(* CODESYS project ETML_DH10.library
   TcLibraryId: TE140x Module Vendor|ETML_DH10|0.0.0.9
   Company: TE140x Module Vendor
   Title: ETML_DH10
   Placeholder: ETML_DH10
   Version: 0.0.0.9

Project tree, tasks and I/O mapping:
  POUs/
    function block FB_ETML_DH10 [ST]: FB_exit, FB_init, nHResult, eInitExceptionHandling, eUpdateExceptionHandling, nExceptionCnt, stActiveException, bInitialized, bExecute
    TcCOM Wrapper/
      function block FB_ETML_DH10_TcCOM_InitStruct [ST]: FB_init, FB_afterinit, Reinit, FB_exit, eObjectState, nHResult, ipTcComObject, ipADI, nTaskOid, nTaskPriority, nTaskCycleTimeNs, nTaskPort, nTaskSortOrder, eTraceLevelMax, eModuleCaller, eCallerVerification, eStepSizeAdaptation, eExecutionSequence, bExecute, eAccessLockState, eInitExceptionHandling, eUpdateExceptionHandling, stModuleBuildInfo, bInitialized, nSkippedExecutionCount, stLibraryInfo, stModuleInfo, stModuleGeneratorInfo, stSimulinkModelInfo, eETML_DH10_P_Sharing, nETML_DH10_P_Definer, stETML_DH10_P, nCycleCount, nExceptionCount, stExceptionInfo
  DUTs/
    data type ST_FB_ETML_DH10_FB_Main
    data type ST_FB_ETML_DH10_FB_exit
    data type ST_FB_ETML_DH10_FB_init
    data type ST_GetSet_HRESULT
    data type E_FpExcptCtrlSetEx
    data type ST_GetSet_E_FpExcptCtrlSetEx
    data type ST_GetSet_ULINT
    data type ST_ExceptionInfo
    data type ST_GetSet_ST_ExceptionInfo
    data type ST_GetSet_BOOL
    data type ST_B_ETML_DH10_T
    data type ST_ExtU_ETML_DH10_T
    data type ST_ExtY_ETML_DH10_T
    data type ST_RT_MODEL_ETML_DH10_T
    data type ST_P_ETML_DH10_T
    data type E_ModuleCaller
    data type E_CallerVerification
    data type E_StepSizeAdaptation
    data type E_ExecutionSequence1
    data type E_FpExcptCtrlSet
    data type ST_TcMatSim_ModuleGeneratorInfo
    data type ST_TcMatSim_SimulinkModelInfo
    data type E_ParameterSharingType
    data type ST_FB_ETML_DH10_TcCOM_InitStruct
    data type ST_FB_ETML_DH10_TcCOM_InitStruct_FB_init
    data type ST_FB_ETML_DH10_TcCOM_InitStruct_FB_afterinit
    data type ST_FB_ETML_DH10_TcCOM_InitStruct_Reinit
    data type ST_FB_ETML_DH10_TcCOM_InitStruct_FB_Main
    data type ST_FB_ETML_DH10_TcCOM_InitStruct_FB_exit
    data type ST_GetSet_TCOM_STATE
    data type ST_GetSet_ITComObject
    data type ST_GetSet_ITcADI
    data type ST_ETML_DH10_U_T
    data type ST_ETML_DH10_Y_T
    data type ST_GetSet_OTCID
    data type ST_GetSet_UDINT
    data type ST_GetSet_UINT
    data type ST_GetSet_TcTraceLevel
    data type ST_GetSet_E_ModuleCaller
    data type ST_GetSet_E_CallerVerification
    data type ST_GetSet_E_StepSizeAdaptation
    data type ST_GetSet_E_ExecutionSequence1
    data type ST_GetSet_E_FpExcptCtrlSet
    data type ST_ModuleBuildInfo
    data type ST_GetSet_ST_ModuleBuildInfo
    data type ST_LibraryInfo
    data type ST_GetSet_ST_LibraryInfo
    data type ST_ModuleInfo
    data type ST_GetSet_ST_ModuleInfo
    data type ST_GetSet_ST_TcMatSim_ModuleGeneratorInfo
    data type ST_GetSet_ST_TcMatSim_SimulinkModelInfo
    data type ST_GetSet_E_ParameterSharingType
    data type ST_GetSet_ST_P_ETML_DH10_T
  Version/
    global variables Global_Version
*)

// DUTs/ST_FB_ETML_DH10_FB_Main
{attribute 'TcIecLibraryType'}
{attribute 'hide'}
TYPE ST_FB_ETML_DH10_FB_Main : 
	STRUCT
		{attribute 'GUID' := '18071995-0000-0000-0000-000000000018'}
		pInst : PVOID;
		result : BOOL;
		 {attribute 'hide'}
		_reserved1 : UINT_24_56;
	END_STRUCT
END_TYPE

// DUTs/ST_FB_ETML_DH10_FB_exit
{attribute 'TcIecLibraryType'}
{attribute 'hide'}
TYPE ST_FB_ETML_DH10_FB_exit : 
	STRUCT
		{attribute 'GUID' := '18071995-0000-0000-0000-000000000018'}
		pInst : PVOID;
		bInCopyCode : BOOL;
		result : BOOL;
		 {attribute 'hide'}
		_reserved1 : UINT_16_48;
	END_STRUCT
END_TYPE

// DUTs/ST_FB_ETML_DH10_FB_init
{attribute 'TcIecLibraryType'}
{attribute 'hide'}
TYPE ST_FB_ETML_DH10_FB_init : 
	STRUCT
		{attribute 'GUID' := '18071995-0000-0000-0000-000000000018'}
		pInst : PVOID;
		bInitRetains : BOOL;
		bInCopyCode : BOOL;
		result : BOOL;
		 {attribute 'hide'}
		_reserved1 : UINT_8_40;
	END_STRUCT
END_TYPE

// DUTs/ST_GetSet_HRESULT
{attribute 'TcIecLibraryType'}
{attribute 'hide'}
TYPE ST_GetSet_HRESULT : 
	STRUCT
		{attribute 'GUID' := '18071995-0000-0000-0000-000000000018'}
		pInst : PVOID;
		{attribute 'GUID' := '18071995-0000-0000-0000-000000000019'}
		nParam : HRESULT;
		 {attribute 'hide'}
		_reserved1 : UINT_0_32;
	END_STRUCT
END_TYPE

// DUTs/E_FpExcptCtrlSetEx
(* Generated from type 'TcMgSdk.FpExcptCtrlSetEx' *)
{attribute 'TcIecLibraryType'}
TYPE E_FpExcptCtrlSetEx : (
	CallerExceptions:=1, 	(* Use the floating point exception settings provided by the caller *)
	ThrowExceptions:=3, 	(* Enable floating point exceptions on invalid operations and divisions by zero *)
	SuppressExceptions:=13, 	(* Disable floating point exceptions. *)
	LogExceptions:=19, 	(* Log exception information. *)
	LogAndHold:=51, 	(* Log exception information and puase execution of the cyclic code after completion of the actual cycle *)
	LogAndCatch:=83, 	(* Log exception information and immediately terminate execution of the cyclic code. Reinitialization is required to restart. *)
	LogAndDump:=147, 	(* Log exception information, create a dump file with detailed exception information and try to continue execution of the cyclic code *)
	LogHoldAndDump:=179, 	(* Log exception information, create a dump file with detailed exception information and puase execution of the cyclic code after completion of the actual cycle *)
	LogCatchAndDump:=211	(* Log exception information, create a dump file with detailed exception information and immediately terminate execution of the cyclic code. Reinitialization is required to restart. *)
) USINT;
END_TYPE

// DUTs/ST_GetSet_E_FpExcptCtrlSetEx
{attribute 'TcIecLibraryType'}
{attribute 'hide'}
TYPE ST_GetSet_E_FpExcptCtrlSetEx : 
	STRUCT
		{attribute 'GUID' := '18071995-0000-0000-0000-000000000018'}
		pInst : PVOID;
		eParam : E_FpExcptCtrlSetEx;
		 {attribute 'hide'}
		_reserved1 : UINT_24_56;
	END_STRUCT
END_TYPE

// DUTs/ST_GetSet_ULINT
{attribute 'TcIecLibraryType'}
{attribute 'hide'}
TYPE ST_GetSet_ULINT : 
	STRUCT
		{attribute 'GUID' := '18071995-0000-0000-0000-000000000018'}
		pInst : PVOID;
		nParam : ULINT;
	END_STRUCT
END_TYPE

// DUTs/ST_ExceptionInfo
(* Generated from type 'TcMgSdk.ExceptionInfo' *)
{attribute 'TcIecLibraryType'}
TYPE ST_ExceptionInfo : 
	STRUCT
		(* Generated from item 'ExceptionCode' *)
		nExceptionCode : DINT;
		(* Generated from item 'TmxName' *)
		{attribute 'GUID' := '18071995-0000-0000-0000-00010000007F'}
		sTmxName : STRING(127);
		(* Generated from item 'TmxVersion' *)
		nTmxVersion : ARRAY [0..3] OF UDINT;
		(* Generated from item 'InstructionAddr' *)
		nInstructionAddr : UDINT;
		(* Generated from item 'ReturnAddr' *)
		nReturnAddr : ARRAY [0..3] OF UDINT;
		(* Generated from item 'DumpCreated' *)
		bDumpCreated : BOOL;
		 {attribute 'hide'}
		_reserved1 : ARRAY [1..3] OF USINT;
	END_STRUCT
END_TYPE

// DUTs/ST_GetSet_ST_ExceptionInfo
{attribute 'TcIecLibraryType'}
{attribute 'hide'}
TYPE ST_GetSet_ST_ExceptionInfo : 
	STRUCT
		{attribute 'GUID' := '18071995-0000-0000-0000-000000000018'}
		pInst : PVOID;
		stParam : ST_ExceptionInfo;
		 {attribute 'hide'}
		_reserved1 : UINT_0_32;
	END_STRUCT
END_TYPE

// DUTs/ST_GetSet_BOOL
{attribute 'TcIecLibraryType'}
{attribute 'hide'}
TYPE ST_GetSet_BOOL : 
	STRUCT
		{attribute 'GUID' := '18071995-0000-0000-0000-000000000018'}
		pInst : PVOID;
		bParam : BOOL;
		 {attribute 'hide'}
		_reserved1 : UINT_24_56;
	END_STRUCT
END_TYPE

// DUTs/ST_B_ETML_DH10_T
(* Generated from type 'B_ETML_DH10_T' *)
{attribute 'TcIecLibraryType'}
TYPE ST_B_ETML_DH10_T : 
	STRUCT
		(* Generated from item 'Sum4' *)
		fSum4 : LREAL;
		(* Generated from item 'Sum5' *)
		fSum5 : LREAL;
		(* Generated from item 'Sum4_g' *)
		fSum4_g : LREAL;
		(* Generated from item 'Sum5_o' *)
		fSum5_o : LREAL;
		(* Generated from item 'Sum4_k' *)
		fSum4_k : LREAL;
		(* Generated from item 'Sum5_c' *)
		fSum5_c : LREAL;
		(* Generated from item 'Sum4_n' *)
		fSum4_n : LREAL;
		(* Generated from item 'Sum5_m' *)
		fSum5_m : LREAL;
		(* Generated from item 'Sum4_c' *)
		fSum4_c : LREAL;
		(* Generated from item 'Sum5_l' *)
		fSum5_l : LREAL;
		(* Generated from item 'Sum4_j' *)
		fSum4_j : LREAL;
		(* Generated from item 'Sum5_p' *)
		fSum5_p : LREAL;
		(* Generated from item 'Sum4_nw' *)
		fSum4_nw : LREAL;
		(* Generated from item 'Sum5_d' *)
		fSum5_d : LREAL;
		(* Generated from item 'Sum4_gt' *)
		fSum4_gt : LREAL;
		(* Generated from item 'Sum5_ob' *)
		fSum5_ob : LREAL;
		(* Generated from item 'q' *)
		fq : LREAL;
		(* Generated from item 'q_g' *)
		fq_g : LREAL;
		(* Generated from item 'q_gi' *)
		fq_gi : LREAL;
		(* Generated from item 'UnaryMinus' *)
		fUnaryMinus : LREAL;
		(* Generated from item 'UnaryMinus_n' *)
		fUnaryMinus_n : LREAL;
		(* Generated from item 'UnaryMinus_o' *)
		fUnaryMinus_o : LREAL;
		(* Generated from item 'UnaryMinus_k' *)
		fUnaryMinus_k : LREAL;
		(* Generated from item 'UnaryMinus_f' *)
		fUnaryMinus_f : LREAL;
		(* Generated from item 'UnaryMinus_l' *)
		fUnaryMinus_l : LREAL;
		(* Generated from item 'UnaryMinus_g' *)
		fUnaryMinus_g : LREAL;
		(* Generated from item 'UnaryMinus_d' *)
		fUnaryMinus_d : LREAL;
		(* Generated from item 's' *)
		fs : LREAL;
		(* Generated from item 's_m' *)
		fs_m : LREAL;
		(* Generated from item 's_h' *)
		fs_h : LREAL;
		(* Generated from item 's_e' *)
		fs_e : LREAL;
		(* Generated from item 's_c' *)
		fs_c : LREAL;
		(* Generated from item 's_l' *)
		fs_l : LREAL;
		(* Generated from item 's_d' *)
		fs_d : LREAL;
		(* Generated from item 's_du' *)
		fs_du : LREAL;
		(* Generated from item 'u' *)
		fu : LREAL;
		(* Generated from item 'Add5' *)
		fAdd5 : LREAL;
		(* Generated from item 'Product4' *)
		fProduct4 : LREAL;
		(* Generated from item 'u_c' *)
		fu_c : LREAL;
		(* Generated from item 'Add5_m' *)
		fAdd5_m : LREAL;
		(* Generated from item 'Product4_p' *)
		fProduct4_p : LREAL;
		(* Generated from item 'u_a' *)
		fu_a : LREAL;
		(* Generated from item 'Add5_j' *)
		fAdd5_j : LREAL;
		(* Generated from item 'Product4_g' *)
		fProduct4_g : LREAL;
		(* Generated from item 'u_l' *)
		fu_l : LREAL;
		(* Generated from item 'Add5_b' *)
		fAdd5_b : LREAL;
		(* Generated from item 'u_m' *)
		fu_m : LREAL;
		(* Generated from item 'Product4_c' *)
		fProduct4_c : LREAL;
		(* Generated from item 'u_o' *)
		fu_o : LREAL;
		(* Generated from item 'Product4_k' *)
		fProduct4_k : LREAL;
		(* Generated from item 'u_g' *)
		fu_g : LREAL;
		(* Generated from item 'Product4_d' *)
		fProduct4_d : LREAL;
		(* Generated from item 'u_p' *)
		fu_p : LREAL;
		(* Generated from item 'Add5_bw' *)
		fAdd5_bw : LREAL;
		(* Generated from item 'Product4_h' *)
		fProduct4_h : LREAL;
		(* Generated from item 'Product1' *)
		fProduct1 : LREAL;
		(* Generated from item 'Product1_e' *)
		fProduct1_e : LREAL;
		(* Generated from item 'Sum2' *)
		fSum2 : LREAL;
		(* Generated from item 'Product1_m' *)
		fProduct1_m : LREAL;
		(* Generated from item 'Sum2_i' *)
		fSum2_i : LREAL;
		(* Generated from item 'Product1_m4' *)
		fProduct1_m4 : LREAL;
		(* Generated from item 'Sum2_j' *)
		fSum2_j : LREAL;
		(* Generated from item 'Product1_f' *)
		fProduct1_f : LREAL;
		(* Generated from item 'UnitDelay2' *)
		fUnitDelay2 : LREAL;
		(* Generated from item 'Product1_l' *)
		fProduct1_l : LREAL;
		(* Generated from item 'UnitDelay2_p' *)
		fUnitDelay2_p : LREAL;
		(* Generated from item 'Product1_a' *)
		fProduct1_a : LREAL;
		(* Generated from item 'UnitDelay2_i' *)
		fUnitDelay2_i : LREAL;
		(* Generated from item 'Product1_o' *)
		fProduct1_o : LREAL;
		(* Generated from item 'Product3' *)
		fProduct3 : LREAL;
		(* Generated from item 'UnitDelay2_l' *)
		fUnitDelay2_l : LREAL;
		(* Generated from item 'Product3_e' *)
		fProduct3_e : LREAL;
		(* Generated from item 'Product3_j' *)
		fProduct3_j : LREAL;
		(* Generated from item 'Product3_a' *)
		fProduct3_a : LREAL;
		(* Generated from item 'Product3_c' *)
		fProduct3_c : LREAL;
		(* Generated from item 'UnitDelay2_k' *)
		fUnitDelay2_k : LREAL;
		(* Generated from item 'Product4_f' *)
		fProduct4_f : LREAL;
		(* Generated from item 'Product3_i' *)
		fProduct3_i : LREAL;
		(* Generated from item 'Product3_o' *)
		fProduct3_o : LREAL;
		(* Generated from item 'Product3_ao' *)
		fProduct3_ao : LREAL;
		(* Generated from item 'RelationalOperator' *)
		bRelationalOperator : BOOL;
		 {attribute 'hide'}
		_reserved1 : ARRAY [1..7] OF USINT;
	END_STRUCT
END_TYPE

// DUTs/ST_ExtU_ETML_DH10_T
(* Generated from type 'ExtU_ETML_DH10_T' *)
{attribute 'TcIecLibraryType'}
TYPE ST_ExtU_ETML_DH10_T : 
	STRUCT
		(* Generated from item 'OffsetLeft' *)
		fOffsetLeft : LREAL;
		(* Generated from item 'OffsetRight' *)
		fOffsetRight : LREAL;
	END_STRUCT
END_TYPE

// DUTs/ST_ExtY_ETML_DH10_T
(* Generated from type 'ExtY_ETML_DH10_T' *)
{attribute 'TcIecLibraryType'}
TYPE ST_ExtY_ETML_DH10_T : 
	STRUCT
		(* Generated from item 'CurrentAngleLeft' *)
		fCurrentAngleLeft : LREAL;
		(* Generated from item 'CurrentAngleRight' *)
		fCurrentAngleRight : LREAL;
	END_STRUCT
END_TYPE

// DUTs/ST_RT_MODEL_ETML_DH10_T
(* Generated from type 'RT_MODEL_ETML_DH10_T' *)
{attribute 'TcIecLibraryType'}
TYPE ST_RT_MODEL_ETML_DH10_T : 
	STRUCT
		errorStatus : POINTER TO SINT;
		blockIO : POINTER TO ST_B_ETML_DH10_T;
		inputs : POINTER TO ST_ExtU_ETML_DH10_T;
		outputs : POINTER TO ST_ExtY_ETML_DH10_T;
	END_STRUCT
END_TYPE

// DUTs/ST_P_ETML_DH10_T
(* Generated from type 'P_ETML_DH10_T' *)
{attribute 'TcIecLibraryType'}
TYPE ST_P_ETML_DH10_T : 
	STRUCT
		(* Generated from item 'ETML_gain_left' *)
		fETML_gain_left : LREAL;
		(* Generated from item 'ETML_gain_right' *)
		fETML_gain_right : LREAL;
		(* Generated from item 'ETML_power_constant' *)
		fETML_power_constant : LREAL;
		(* Generated from item 'f_ETML_notch_main_1' *)
		ff_ETML_notch_main_1 : LREAL;
		(* Generated from item 'f_ETML_notch_main_2' *)
		ff_ETML_notch_main_2 : LREAL;
		(* Generated from item 'f_ETML_notch_main_3' *)
		ff_ETML_notch_main_3 : LREAL;
		(* Generated from item 'f_ETML_notch_main_4' *)
		ff_ETML_notch_main_4 : LREAL;
		(* Generated from item 'notch_damp' *)
		fnotch_damp : LREAL;
		(* Generated from item 'notch_gmin' *)
		fnotch_gmin : LREAL;
		(* Generated from item 'enable_ETML_main_notch_1' *)
		benable_ETML_main_notch_1 : BOOL;
		(* Generated from item 'enable_ETML_main_notch_2' *)
		benable_ETML_main_notch_2 : BOOL;
		(* Generated from item 'enable_ETML_main_notch_3' *)
		benable_ETML_main_notch_3 : BOOL;
		(* Generated from item 'enable_ETML_main_notch_4' *)
		benable_ETML_main_notch_4 : BOOL;
		 {attribute 'hide'}
		_reserved1 : UDINT;
		(* Generated from item 'Constant2_Value' *)
		fConstant2_Value : LREAL;
		(* Generated from item 'Constant_Value' *)
		fConstant_Value : LREAL;
		(* Generated from item 'tau_Gain' *)
		ftau_Gain : LREAL;
		(* Generated from item 'Bias_Bias' *)
		fBias_Bias : LREAL;
		(* Generated from item 'two_Gain' *)
		ftwo_Gain : LREAL;
		(* Generated from item 'one_Gain' *)
		fone_Gain : LREAL;
		(* Generated from item 'UnitDelay1_InitialCondition' *)
		fUnitDelay1_InitialCondition : LREAL;
		(* Generated from item 'tau_Gain_n' *)
		ftau_Gain_n : LREAL;
		(* Generated from item 'Bias_Bias_e' *)
		fBias_Bias_e : LREAL;
		(* Generated from item 'two_Gain_i' *)
		ftwo_Gain_i : LREAL;
		(* Generated from item 'one_Gain_k' *)
		fone_Gain_k : LREAL;
		(* Generated from item 'UnitDelay1_InitialCondition_p' *)
		fUnitDelay1_InitialCondition_p : LREAL;
		(* Generated from item 'tau_Gain_j' *)
		ftau_Gain_j : LREAL;
		(* Generated from item 'Bias_Bias_h' *)
		fBias_Bias_h : LREAL;
		(* Generated from item 'two_Gain_b' *)
		ftwo_Gain_b : LREAL;
		(* Generated from item 'one_Gain_e' *)
		fone_Gain_e : LREAL;
		(* Generated from item 'UnitDelay1_InitialCondition_b' *)
		fUnitDelay1_InitialCondition_b : LREAL;
		(* Generated from item 'tau_Gain_k' *)
		ftau_Gain_k : LREAL;
		(* Generated from item 'Bias_Bias_a' *)
		fBias_Bias_a : LREAL;
		(* Generated from item 'two_Gain_h' *)
		ftwo_Gain_h : LREAL;
		(* Generated from item 'one_Gain_ea' *)
		fone_Gain_ea : LREAL;
		(* Generated from item 'UnitDelay1_InitialCondition_d' *)
		fUnitDelay1_InitialCondition_d : LREAL;
		(* Generated from item 'Left_UpperSat' *)
		fLeft_UpperSat : LREAL;
		(* Generated from item 'Left_LowerSat' *)
		fLeft_LowerSat : LREAL;
		(* Generated from item 'tau_Gain_l' *)
		ftau_Gain_l : LREAL;
		(* Generated from item 'Bias_Bias_j' *)
		fBias_Bias_j : LREAL;
		(* Generated from item 'two_Gain_o' *)
		ftwo_Gain_o : LREAL;
		(* Generated from item 'one_Gain_o' *)
		fone_Gain_o : LREAL;
		(* Generated from item 'UnitDelay1_InitialCondition_j' *)
		fUnitDelay1_InitialCondition_j : LREAL;
		(* Generated from item 'tau_Gain_f' *)
		ftau_Gain_f : LREAL;
		(* Generated from item 'Bias_Bias_b' *)
		fBias_Bias_b : LREAL;
		(* Generated from item 'two_Gain_c' *)
		ftwo_Gain_c : LREAL;
		(* Generated from item 'one_Gain_l' *)
		fone_Gain_l : LREAL;
		(* Generated from item 'UnitDelay1_InitialCondition_a' *)
		fUnitDelay1_InitialCondition_a : LREAL;
		(* Generated from item 'tau_Gain_lc' *)
		ftau_Gain_lc : LREAL;
		(* Generated from item 'Bias_Bias_i' *)
		fBias_Bias_i : LREAL;
		(* Generated from item 'two_Gain_m' *)
		ftwo_Gain_m : LREAL;
		(* Generated from item 'one_Gain_ef' *)
		fone_Gain_ef : LREAL;
		(* Generated from item 'UnitDelay1_InitialCondition_d5' *)
		fUnitDelay1_InitialCondition_d5 : LREAL;
		(* Generated from item 'tau_Gain_e' *)
		ftau_Gain_e : LREAL;
		(* Generated from item 'Bias_Bias_l' *)
		fBias_Bias_l : LREAL;
		(* Generated from item 'two_Gain_it' *)
		ftwo_Gain_it : LREAL;
		(* Generated from item 'one_Gain_a' *)
		fone_Gain_a : LREAL;
		(* Generated from item 'UnitDelay1_InitialCondition_l' *)
		fUnitDelay1_InitialCondition_l : LREAL;
		(* Generated from item 'Right_UpperSat' *)
		fRight_UpperSat : LREAL;
		(* Generated from item 'Right_LowerSat' *)
		fRight_LowerSat : LREAL;
		(* Generated from item 'Bias1_Bias' *)
		fBias1_Bias : LREAL;
		(* Generated from item 'Gain_Gain' *)
		fGain_Gain : LREAL;
		(* Generated from item 'UnitDelay2_InitialCondition' *)
		fUnitDelay2_InitialCondition : LREAL;
		(* Generated from item 'Bias1_Bias_b' *)
		fBias1_Bias_b : LREAL;
		(* Generated from item 'Gain_Gain_g' *)
		fGain_Gain_g : LREAL;
		(* Generated from item 'UnitDelay2_InitialCondition_p' *)
		fUnitDelay2_InitialCondition_p : LREAL;
		(* Generated from item 'Bias1_Bias_n' *)
		fBias1_Bias_n : LREAL;
		(* Generated from item 'Gain_Gain_k' *)
		fGain_Gain_k : LREAL;
		(* Generated from item 'UnitDelay2_InitialCondition_o' *)
		fUnitDelay2_InitialCondition_o : LREAL;
		(* Generated from item 'Bias1_Bias_c' *)
		fBias1_Bias_c : LREAL;
		(* Generated from item 'Gain_Gain_e' *)
		fGain_Gain_e : LREAL;
		(* Generated from item 'UnitDelay2_InitialCondition_f' *)
		fUnitDelay2_InitialCondition_f : LREAL;
		(* Generated from item 'Bias1_Bias_l' *)
		fBias1_Bias_l : LREAL;
		(* Generated from item 'Gain_Gain_ey' *)
		fGain_Gain_ey : LREAL;
		(* Generated from item 'UnitDelay2_InitialCondition_k' *)
		fUnitDelay2_InitialCondition_k : LREAL;
		(* Generated from item 'Bias1_Bias_j' *)
		fBias1_Bias_j : LREAL;
		(* Generated from item 'Gain_Gain_ky' *)
		fGain_Gain_ky : LREAL;
		(* Generated from item 'UnitDelay2_InitialCondition_l' *)
		fUnitDelay2_InitialCondition_l : LREAL;
		(* Generated from item 'Bias1_Bias_d' *)
		fBias1_Bias_d : LREAL;
		(* Generated from item 'Gain_Gain_f' *)
		fGain_Gain_f : LREAL;
		(* Generated from item 'UnitDelay2_InitialCondition_n' *)
		fUnitDelay2_InitialCondition_n : LREAL;
		(* Generated from item 'Bias1_Bias_cn' *)
		fBias1_Bias_cn : LREAL;
		(* Generated from item 'Gain_Gain_h' *)
		fGain_Gain_h : LREAL;
		(* Generated from item 'UnitDelay2_InitialCondition_i' *)
		fUnitDelay2_InitialCondition_i : LREAL;
	END_STRUCT
END_TYPE

// DUTs/E_ModuleCaller
(* Generated from type 'TcMgSdk.ModuleCaller' *)
{attribute 'TcIecLibraryType'}
TYPE E_ModuleCaller : (
	CyclicTask:=0, 	(* Add to the specified cyclic caller tasks. *)
	Module:=1	(* Don't add to cyclic callers. The module can be called from other TwinCAT modules (e. g. a PLC). *)
) DINT;
END_TYPE

// DUTs/E_CallerVerification
(* Generated from type 'TcMgSdk.CallerVerification' *)
{attribute 'TcIecLibraryType'}
TYPE E_CallerVerification : (
	Default:=0, 	(* Verify the caller task only if the "ModuleCaller" parameter is set to "Module" but not when added to cyclic caller tasks. *)
	Always:=1, 	(* Always verify the caller context to prevent concurrent execution of model code and corresponding DataArea mappings. *)
	Never:=2	(* Skip caller verification to reduce execution times. *)
) DINT;
END_TYPE

// DUTs/E_StepSizeAdaptation
(* Generated from type 'TcMgSdk.StepSizeAdaptation' *)
{attribute 'TcIecLibraryType'}
TYPE E_StepSizeAdaptation : (
	RequireMatchingTaskCycleTime:=0, 	(* Don't accept task cycle times other than the Simulink step sizes. *)
	UseTaskCycleTime:=1, 	(* Adapt the Smulink step sizes to the task cycle times. *)
	UseModelStepSize:=2	(* Keep the Smulink step sizes, independent of the callers cycle time. *)
) DINT;
END_TYPE

// DUTs/E_ExecutionSequence1
(* Generated from type 'TcMgSdk.ExecutionSequence1' *)
{attribute 'TcIecLibraryType'}
TYPE E_ExecutionSequence1 : (
	UpdateBeforeOutputMapping:=0, 	(* Input mapping -> State and output update -> Output mapping -> ADS processing *)
	IoAtTaskBegin:=1	(* Input mapping -> Code execution -> Output update -> ADS processing *)
) DINT;
END_TYPE

// DUTs/E_FpExcptCtrlSet
(* Generated from type 'TcMgSdk.FpExcptCtrlSet' *)
{attribute 'TcIecLibraryType'}
TYPE E_FpExcptCtrlSet : (
	CallerExceptions:=1, 	(* Use the floating point exception settings provided by the caller *)
	ThrowExceptions:=3, 	(* Enable floating point exceptions on invalid operations and divisions by zero *)
	SuppressExceptions:=5	(* Disable floating point exceptions. *)
) USINT;
END_TYPE

// DUTs/ST_TcMatSim_ModuleGeneratorInfo
(* Generated from type 'TcMatSim.ModuleGeneratorInfo' *)
{attribute 'TcIecLibraryType'}
TYPE ST_TcMatSim_ModuleGeneratorInfo : 
	STRUCT
		(* Generated from item 'MatlabVersion' *)
		nMatlabVersion : ARRAY [0..3] OF UDINT;
		(* Generated from item 'TE140xVersion' *)
		nTE140xVersion : ARRAY [0..3] OF UDINT;
	END_STRUCT
END_TYPE

// DUTs/ST_TcMatSim_SimulinkModelInfo
(* Generated from type 'TcMatSim.SimulinkModelInfo' *)
{attribute 'TcIecLibraryType'}
TYPE ST_TcMatSim_SimulinkModelInfo : 
	STRUCT
		(* Generated from item 'ModelName' *)
		{attribute 'GUID' := '18071995-0000-0000-0000-00010000007F'}
		sModelName : STRING(127);
		(* Generated from item 'SimulinkVersion' *)
		nSimulinkVersion : ARRAY [0..3] OF UDINT;
		(* Generated from item 'ModelVersion' *)
		nModelVersion : ARRAY [0..3] OF UDINT;
		(* Generated from item 'ModelChecksum' *)
		nModelChecksum : ARRAY [0..3] OF UDINT;
	END_STRUCT
END_TYPE

// DUTs/E_ParameterSharingType
(* Generated from type 'ParameterSharingType' *)
{attribute 'TcIecLibraryType'}
TYPE E_ParameterSharingType : (
	Define:=0, 	(* This module instance defines the parameter values for all further instances of this module class. Exactly one instance of this module class must use this option. *)
	Inherit:=1	(* This module instance inherits the parameter values from the instance of this module class configured to "Define" the parameter values. Model parameters configured at this instsance are ignored. *)
) DINT;
END_TYPE

// DUTs/ST_FB_ETML_DH10_TcCOM_InitStruct
{attribute 'TcIecLibraryType'}
TYPE ST_FB_ETML_DH10_TcCOM_InitStruct : 
	STRUCT
		{attribute 'GUID' := '18071995-0000-0000-0000-000000000061'}
		eObjState : TCOM_STATE := TCOM_STATE.TCOM_STATE_OP;
		{attribute 'GUID' := '18071995-0000-0000-0000-00010000007F'}
		sObjName : STRING(127);
		{attribute 'GUID' := '18071995-0000-0000-0000-00000000000F'}
		nOid : OTCID := 4294967295;
		{attribute 'GUID' := '18071995-0000-0000-0000-00000000000F'}
		nTaskOid : OTCID;
		nTaskSortOrder : UDINT;
		{attribute 'GUID' := '8007AE3B-86BB-40F2-B385-EF87FCC239A4'}
		eTraceLevelMax : TcTraceLevel := TcTraceLevel.tlInfo;
		eModuleCaller : E_ModuleCaller := E_ModuleCaller.CyclicTask;
		eCallerVerification : E_CallerVerification := E_CallerVerification.Default;
		eStepSizeAdaptation : E_StepSizeAdaptation := E_StepSizeAdaptation.RequireMatchingTaskCycleTime;
		eExecutionSequence : E_ExecutionSequence1 := E_ExecutionSequence1.UpdateBeforeOutputMapping;
		bExecute : BOOL := TRUE;
		 {attribute 'hide'}
		_reserved1 : ARRAY [1..3] OF USINT;
		{attribute 'GUID' := '18071995-0000-0000-0000-000000000061'}
		eAccessLockState : TCOM_STATE := TCOM_STATE.TCOM_STATE_OP;
		eInitExceptionHandling : E_FpExcptCtrlSet := E_FpExcptCtrlSet.CallerExceptions;
		eUpdateExceptionHandling : E_FpExcptCtrlSetEx := E_FpExcptCtrlSetEx.CallerExceptions;
		 {attribute 'hide'}
		_reserved2 : UINT;
		stModuleGeneratorInfo : ST_TcMatSim_ModuleGeneratorInfo;
		stSimulinkModelInfo : ST_TcMatSim_SimulinkModelInfo;
		eETML_DH10_P_Sharing : E_ParameterSharingType := E_ParameterSharingType.Define;
		 {attribute 'hide'}
		_reserved3 : UDINT;
		stETML_DH10_P : ST_P_ETML_DH10_T := (fETML_gain_left := 16.91503741, fETML_gain_right := 16.91503741, fETML_power_constant := 0.46047809, ff_ETML_notch_main_1 := 0, ff_ETML_notch_main_2 := 0, ff_ETML_notch_main_3 := 0, ff_ETML_notch_main_4 := 0, fnotch_damp := 0.3, fnotch_gmin := 0.1, benable_ETML_main_notch_1 := FALSE, benable_ETML_main_notch_2 := FALSE, benable_ETML_main_notch_3 := FALSE, benable_ETML_main_notch_4 := FALSE, fConstant2_Value := 45, fConstant_Value := 0, ftau_Gain := 0.003, fBias_Bias := 1, ftwo_Gain := 2, fone_Gain := 1, fUnitDelay1_InitialCondition := 0, ftau_Gain_n := 0.003, fBias_Bias_e := 1, ftwo_Gain_i := 2, fone_Gain_k := 1, fUnitDelay1_InitialCondition_p := 0, ftau_Gain_j := 0.003, fBias_Bias_h := 1, ftwo_Gain_b := 2, fone_Gain_e := 1, fUnitDelay1_InitialCondition_b := 0, ftau_Gain_k := 0.003, fBias_Bias_a := 1, ftwo_Gain_h := 2, fone_Gain_ea := 1, fUnitDelay1_InitialCondition_d := 0, fLeft_UpperSat := 90, fLeft_LowerSat := 0, ftau_Gain_l := 0.003, fBias_Bias_j := 1, ftwo_Gain_o := 2, fone_Gain_o := 1, fUnitDelay1_InitialCondition_j := 0, ftau_Gain_f := 0.003, fBias_Bias_b := 1, ftwo_Gain_c := 2, fone_Gain_l := 1, fUnitDelay1_InitialCondition_a := 0, ftau_Gain_lc := 0.003, fBias_Bias_i := 1, ftwo_Gain_m := 2, fone_Gain_ef := 1, fUnitDelay1_InitialCondition_d5 := 0, ftau_Gain_e := 0.003, fBias_Bias_l := 1, ftwo_Gain_it := 2, fone_Gain_a := 1, fUnitDelay1_InitialCondition_l := 0, fRight_UpperSat := 90, fRight_LowerSat := 0, fBias1_Bias := 1, fGain_Gain := 2, fUnitDelay2_InitialCondition := 0, fBias1_Bias_b := 1, fGain_Gain_g := 2, fUnitDelay2_InitialCondition_p := 0, fBias1_Bias_n := 1, fGain_Gain_k := 2, fUnitDelay2_InitialCondition_o := 0, fBias1_Bias_c := 1, fGain_Gain_e := 2, fUnitDelay2_InitialCondition_f := 0, fBias1_Bias_l := 1, fGain_Gain_ey := 2, fUnitDelay2_InitialCondition_k := 0, fBias1_Bias_j := 1, fGain_Gain_ky := 2, fUnitDelay2_InitialCondition_l := 0, fBias1_Bias_d := 1, fGain_Gain_f := 2, fUnitDelay2_InitialCondition_n := 0, fBias1_Bias_cn := 1, fGain_Gain_h := 2, fUnitDelay2_InitialCondition_i := 0);
	END_STRUCT
END_TYPE

// DUTs/ST_FB_ETML_DH10_TcCOM_InitStruct_FB_init
{attribute 'TcIecLibraryType'}
{attribute 'hide'}
TYPE ST_FB_ETML_DH10_TcCOM_InitStruct_FB_init : 
	STRUCT
		{attribute 'GUID' := '18071995-0000-0000-0000-000000000018'}
		pInst : PVOID;
		bInitRetains : BOOL;
		bInCopyCode : BOOL;
		 {attribute 'hide'}
		_reserved1 : UINT_16_48;
		stInit : REFERENCE TO ST_FB_ETML_DH10_TcCOM_InitStruct;
		result : BOOL;
		 {attribute 'hide'}
		_reserved2 : UINT_24_56;
	END_STRUCT
END_TYPE

// DUTs/ST_FB_ETML_DH10_TcCOM_InitStruct_FB_afterinit
{attribute 'TcIecLibraryType'}
{attribute 'hide'}
TYPE ST_FB_ETML_DH10_TcCOM_InitStruct_FB_afterinit : 
	STRUCT
		{attribute 'GUID' := '18071995-0000-0000-0000-000000000018'}
		pInst : PVOID;
		result : BOOL;
		 {attribute 'hide'}
		_reserved1 : UINT_24_56;
	END_STRUCT
END_TYPE

// DUTs/ST_FB_ETML_DH10_TcCOM_InitStruct_Reinit
{attribute 'TcIecLibraryType'}
{attribute 'hide'}
TYPE ST_FB_ETML_DH10_TcCOM_InitStruct_Reinit : 
	STRUCT
		{attribute 'GUID' := '18071995-0000-0000-0000-000000000018'}
		pInst : PVOID;
		stReInit : ST_FB_ETML_DH10_TcCOM_InitStruct;
		result : BOOL;
		 {attribute 'hide'}
		_reserved1 : ARRAY [1..7] OF USINT;
	END_STRUCT
END_TYPE

// DUTs/ST_FB_ETML_DH10_TcCOM_InitStruct_FB_Main
{attribute 'TcIecLibraryType'}
{attribute 'hide'}
TYPE ST_FB_ETML_DH10_TcCOM_InitStruct_FB_Main : 
	STRUCT
		{attribute 'GUID' := '18071995-0000-0000-0000-000000000018'}
		pInst : PVOID;
		result : BOOL;
		 {attribute 'hide'}
		_reserved1 : UINT_24_56;
	END_STRUCT
END_TYPE

// DUTs/ST_FB_ETML_DH10_TcCOM_InitStruct_FB_exit
{attribute 'TcIecLibraryType'}
{attribute 'hide'}
TYPE ST_FB_ETML_DH10_TcCOM_InitStruct_FB_exit : 
	STRUCT
		{attribute 'GUID' := '18071995-0000-0000-0000-000000000018'}
		pInst : PVOID;
		bInCopyCode : BOOL;
		result : BOOL;
		 {attribute 'hide'}
		_reserved1 : UINT_16_48;
	END_STRUCT
END_TYPE

// DUTs/ST_GetSet_TCOM_STATE
{attribute 'TcIecLibraryType'}
{attribute 'hide'}
TYPE ST_GetSet_TCOM_STATE : 
	STRUCT
		{attribute 'GUID' := '18071995-0000-0000-0000-000000000018'}
		pInst : PVOID;
		{attribute 'GUID' := '18071995-0000-0000-0000-000000000061'}
		eParam : TCOM_STATE;
		 {attribute 'hide'}
		_reserved1 : UINT_0_32;
	END_STRUCT
END_TYPE

// DUTs/ST_GetSet_ITComObject
{attribute 'TcIecLibraryType'}
{attribute 'hide'}
TYPE ST_GetSet_ITComObject : 
	STRUCT
		{attribute 'GUID' := '18071995-0000-0000-0000-000000000018'}
		pInst : PVOID;
		{attribute 'GUID' := '00000012-0000-0000-E000-000000000064'}
		ipParam : ITComObject;
	END_STRUCT
END_TYPE

// DUTs/ST_GetSet_ITcADI
{attribute 'TcIecLibraryType'}
{attribute 'hide'}
TYPE ST_GetSet_ITcADI : 
	STRUCT
		{attribute 'GUID' := '18071995-0000-0000-0000-000000000018'}
		pInst : PVOID;
		{attribute 'GUID' := '03000012-0000-0000-E000-000000000064'}
		ipParam : ITcADI;
	END_STRUCT
END_TYPE

// DUTs/ST_ETML_DH10_U_T
(* Generated from type 'ETML_DH10_U_T' *)
{attribute 'TcIecLibraryType'}
TYPE ST_ETML_DH10_U_T : 
	STRUCT
		(* Generated from item 'OffsetLeft' *)
		fOffsetLeft : LREAL;
		(* Generated from item 'OffsetRight' *)
		fOffsetRight : LREAL;
	END_STRUCT
END_TYPE

// DUTs/ST_ETML_DH10_Y_T
(* Generated from type 'ETML_DH10_Y_T' *)
{attribute 'TcIecLibraryType'}
TYPE ST_ETML_DH10_Y_T : 
	STRUCT
		(* Generated from item 'CurrentAngleLeft' *)
		fCurrentAngleLeft : LREAL;
		(* Generated from item 'CurrentAngleRight' *)
		fCurrentAngleRight : LREAL;
	END_STRUCT
END_TYPE

// DUTs/ST_GetSet_OTCID
{attribute 'TcIecLibraryType'}
{attribute 'hide'}
TYPE ST_GetSet_OTCID : 
	STRUCT
		{attribute 'GUID' := '18071995-0000-0000-0000-000000000018'}
		pInst : PVOID;
		{attribute 'GUID' := '18071995-0000-0000-0000-00000000000F'}
		nParam : OTCID;
		 {attribute 'hide'}
		_reserved1 : UINT_0_32;
	END_STRUCT
END_TYPE

// DUTs/ST_GetSet_UDINT
{attribute 'TcIecLibraryType'}
{attribute 'hide'}
TYPE ST_GetSet_UDINT : 
	STRUCT
		{attribute 'GUID' := '18071995-0000-0000-0000-000000000018'}
		pInst : PVOID;
		nParam : UDINT;
		 {attribute 'hide'}
		_reserved1 : UINT_0_32;
	END_STRUCT
END_TYPE

// DUTs/ST_GetSet_UINT
{attribute 'TcIecLibraryType'}
{attribute 'hide'}
TYPE ST_GetSet_UINT : 
	STRUCT
		{attribute 'GUID' := '18071995-0000-0000-0000-000000000018'}
		pInst : PVOID;
		nParam : UINT;
		 {attribute 'hide'}
		_reserved1 : UINT_16_48;
	END_STRUCT
END_TYPE

// DUTs/ST_GetSet_TcTraceLevel
{attribute 'TcIecLibraryType'}
{attribute 'hide'}
TYPE ST_GetSet_TcTraceLevel : 
	STRUCT
		{attribute 'GUID' := '18071995-0000-0000-0000-000000000018'}
		pInst : PVOID;
		{attribute 'GUID' := '8007AE3B-86BB-40F2-B385-EF87FCC239A4'}
		eParam : TcTraceLevel;
		 {attribute 'hide'}
		_reserved1 : UINT_0_32;
	END_STRUCT
END_TYPE

// DUTs/ST_GetSet_E_ModuleCaller
{attribute 'TcIecLibraryType'}
{attribute 'hide'}
TYPE ST_GetSet_E_ModuleCaller : 
	STRUCT
		{attribute 'GUID' := '18071995-0000-0000-0000-000000000018'}
		pInst : PVOID;
		eParam : E_ModuleCaller;
		 {attribute 'hide'}
		_reserved1 : UINT_0_32;
	END_STRUCT
END_TYPE

// DUTs/ST_GetSet_E_CallerVerification
{attribute 'TcIecLibraryType'}
{attribute 'hide'}
TYPE ST_GetSet_E_CallerVerification : 
	STRUCT
		{attribute 'GUID' := '18071995-0000-0000-0000-000000000018'}
		pInst : PVOID;
		eParam : E_CallerVerification;
		 {attribute 'hide'}
		_reserved1 : UINT_0_32;
	END_STRUCT
END_TYPE

// DUTs/ST_GetSet_E_StepSizeAdaptation
{attribute 'TcIecLibraryType'}
{attribute 'hide'}
TYPE ST_GetSet_E_StepSizeAdaptation : 
	STRUCT
		{attribute 'GUID' := '18071995-0000-0000-0000-000000000018'}
		pInst : PVOID;
		eParam : E_StepSizeAdaptation;
		 {attribute 'hide'}
		_reserved1 : UINT_0_32;
	END_STRUCT
END_TYPE

// DUTs/ST_GetSet_E_ExecutionSequence1
{attribute 'TcIecLibraryType'}
{attribute 'hide'}
TYPE ST_GetSet_E_ExecutionSequence1 : 
	STRUCT
		{attribute 'GUID' := '18071995-0000-0000-0000-000000000018'}
		pInst : PVOID;
		eParam : E_ExecutionSequence1;
		 {attribute 'hide'}
		_reserved1 : UINT_0_32;
	END_STRUCT
END_TYPE

// DUTs/ST_GetSet_E_FpExcptCtrlSet
{attribute 'TcIecLibraryType'}
{attribute 'hide'}
TYPE ST_GetSet_E_FpExcptCtrlSet : 
	STRUCT
		{attribute 'GUID' := '18071995-0000-0000-0000-000000000018'}
		pInst : PVOID;
		eParam : E_FpExcptCtrlSet;
		 {attribute 'hide'}
		_reserved1 : UINT_24_56;
	END_STRUCT
END_TYPE

// DUTs/ST_ModuleBuildInfo
(* Generated from type 'TcMgSdk.ModuleBuildInfo' *)
{attribute 'TcIecLibraryType'}
TYPE ST_ModuleBuildInfo : 
	STRUCT
		(* Generated from item 'TcBuild' *)
		nTcBuild : UDINT;
		(* Generated from item 'TcRevision' *)
		nTcRevision : UDINT;
		(* Generated from item 'Debug' *)
		bDebug : BOOL;
		 {attribute 'hide'}
		_reserved1 : ARRAY [1..3] OF USINT;
	END_STRUCT
END_TYPE

// DUTs/ST_GetSet_ST_ModuleBuildInfo
{attribute 'TcIecLibraryType'}
{attribute 'hide'}
TYPE ST_GetSet_ST_ModuleBuildInfo : 
	STRUCT
		{attribute 'GUID' := '18071995-0000-0000-0000-000000000018'}
		pInst : PVOID;
		stParam : ST_ModuleBuildInfo;
		 {attribute 'hide'}
		_reserved1 : UINT_0_32;
	END_STRUCT
END_TYPE

// DUTs/ST_LibraryInfo
(* Generated from type 'TcMgSdk.LibraryInfo' *)
{attribute 'TcIecLibraryType'}
TYPE ST_LibraryInfo : 
	STRUCT
		(* Generated from item 'FileVersion' *)
		nFileVersion : ARRAY [0..3] OF UDINT;
		(* Generated from item 'ProductVersion' *)
		nProductVersion : ARRAY [0..3] OF UDINT;
		(* Generated from item 'VendorName' *)
		{attribute 'GUID' := '18071995-0000-0000-0000-00010000007F'}
		sVendorName : STRING(127);
		(* Generated from item 'LibraryName' *)
		{attribute 'GUID' := '18071995-0000-0000-0000-00010000007F'}
		sLibraryName : STRING(127);
		(* Generated from item 'LibraryVersion' *)
		nLibraryVersion : ARRAY [0..3] OF UDINT;
		(* Generated from item 'LibraryId' *)
		{attribute 'GUID' := '18071995-0000-0000-0000-00010000007F'}
		sLibraryId : STRING(127);
		(* Generated from item 'LibraryGUID' *)
		{attribute 'GUID' := '18071995-0000-0000-0000-000000000024'}
		nLibraryGUID : CLSID;
		(* Generated from item 'TcSdkVersion' *)
		nTcSdkVersion : ARRAY [0..3] OF UDINT;
		(* Generated from item 'Compiler' *)
		{attribute 'GUID' := '18071995-0000-0000-0000-00010000007F'}
		sCompiler : STRING(127);
		(* Generated from item 'Debug' *)
		bDebug : BOOL;
		 {attribute 'hide'}
		_reserved1 : ARRAY [1..7] OF USINT;
	END_STRUCT
END_TYPE

// DUTs/ST_GetSet_ST_LibraryInfo
{attribute 'TcIecLibraryType'}
{attribute 'hide'}
TYPE ST_GetSet_ST_LibraryInfo : 
	STRUCT
		{attribute 'GUID' := '18071995-0000-0000-0000-000000000018'}
		pInst : PVOID;
		stParam : ST_LibraryInfo;
	END_STRUCT
END_TYPE

// DUTs/ST_ModuleInfo
(* Generated from type 'TcMgSdk.ModuleInfo' *)
{attribute 'TcIecLibraryType'}
TYPE ST_ModuleInfo : 
	STRUCT
		(* Generated from item 'ClassName' *)
		{attribute 'GUID' := '18071995-0000-0000-0000-00010000007F'}
		sClassName : STRING(127);
		(* Generated from item 'CommonClassId' *)
		{attribute 'GUID' := '18071995-0000-0000-0000-000000000024'}
		nCommonClassId : CLSID;
		(* Generated from item 'VersionClassId' *)
		{attribute 'GUID' := '18071995-0000-0000-0000-000000000024'}
		nVersionClassId : CLSID;
	END_STRUCT
END_TYPE

// DUTs/ST_GetSet_ST_ModuleInfo
{attribute 'TcIecLibraryType'}
{attribute 'hide'}
TYPE ST_GetSet_ST_ModuleInfo : 
	STRUCT
		{attribute 'GUID' := '18071995-0000-0000-0000-000000000018'}
		pInst : PVOID;
		stParam : ST_ModuleInfo;
	END_STRUCT
END_TYPE

// DUTs/ST_GetSet_ST_TcMatSim_ModuleGeneratorInfo
{attribute 'TcIecLibraryType'}
{attribute 'hide'}
TYPE ST_GetSet_ST_TcMatSim_ModuleGeneratorInfo : 
	STRUCT
		{attribute 'GUID' := '18071995-0000-0000-0000-000000000018'}
		pInst : PVOID;
		stParam : ST_TcMatSim_ModuleGeneratorInfo;
	END_STRUCT
END_TYPE

// DUTs/ST_GetSet_ST_TcMatSim_SimulinkModelInfo
{attribute 'TcIecLibraryType'}
{attribute 'hide'}
TYPE ST_GetSet_ST_TcMatSim_SimulinkModelInfo : 
	STRUCT
		{attribute 'GUID' := '18071995-0000-0000-0000-000000000018'}
		pInst : PVOID;
		stParam : ST_TcMatSim_SimulinkModelInfo;
	END_STRUCT
END_TYPE

// DUTs/ST_GetSet_E_ParameterSharingType
{attribute 'TcIecLibraryType'}
{attribute 'hide'}
TYPE ST_GetSet_E_ParameterSharingType : 
	STRUCT
		{attribute 'GUID' := '18071995-0000-0000-0000-000000000018'}
		pInst : PVOID;
		eParam : E_ParameterSharingType;
		 {attribute 'hide'}
		_reserved1 : UINT_0_32;
	END_STRUCT
END_TYPE

// DUTs/ST_GetSet_ST_P_ETML_DH10_T
{attribute 'TcIecLibraryType'}
{attribute 'hide'}
TYPE ST_GetSet_ST_P_ETML_DH10_T : 
	STRUCT
		{attribute 'GUID' := '18071995-0000-0000-0000-000000000018'}
		pInst : PVOID;
		stParam : ST_P_ETML_DH10_T;
	END_STRUCT
END_TYPE

// Version/Global_Version
{attribute 'TcGenerated'}
// This function has been automatically generated from the project information.
VAR_GLOBAL CONSTANT
	{attribute 'const_non_replaced'}
	{attribute 'linkalways'}
	stLibVersion_ETML_DH10 : ST_LibVersion := (iMajor := 0, iMinor := 0, iBuild := 0, iRevision := 9, nFlags := 0, sVersion := '0.0.0.9');
	{attribute 'const_non_replaced'}
	{attribute 'linkalways'}
	sLibraryId_ETML_DH10 : String := 'TE140x Module Vendor|ETML_DH10|0.0.0.9';
END_VAR

// POUs/FB_ETML_DH10

{attribute 'c++_compatible'}
{attribute 'external_name' := 'FB_ETML_DH10_GUID_51EC76E1_8923_3084_6CCC_B43CA1594E6A'}
{attribute 'TcIecLibraryType'}
{attribute 'reflection'}
FUNCTION_BLOCK FB_ETML_DH10
VAR
	{attribute 'hide'}
	{attribute 'no_copy'}
	{attribute 'GUID' := '18071995-0000-0000-0000-000000000018'}
	m_pData : PVOID;
	{attribute 'TcInitSymbol'}
	{attribute 'GUID' := '8007AE3B-86BB-40F2-B385-EF87FCC239A4'}
	eTraceLevelMax : TcTraceLevel := TcTraceLevel.tlInfo;
	 {attribute 'hide'}
	_reserved1 : UDINT;
	{attribute 'hide'}
	{attribute 'instance-path'}
	{attribute 'noinit'}
	{attribute 'GUID' := '18071995-0000-0000-0000-0001000000FF'}
	sInstancePath : STRING(255);
	{attribute 'hide'}
	{attribute 'noinit'}
	{attribute 'GUID' := '18071995-0000-0000-0000-000000000019'}
	m_HResultLog : HRESULT;
	{attribute 'hide'}
	{attribute 'noinit'}
	{attribute 'GUID' := '18071995-0000-0000-0000-000000000019'}
	m_HResult : HRESULT;
	 {attribute 'hide'}
	_reserved2 : ARRAY [1..184] OF USINT;
	{attribute 'hide'}
	{attribute 'no_copy'}
	m_ExtModeData : ULINT;
END_VAR
VAR_INPUT
	(* Generated from item 'OffsetLeft' *)
	fOffsetLeft : LREAL;
	(* Generated from item 'OffsetRight' *)
	fOffsetRight : LREAL;
END_VAR
VAR_OUTPUT
	(* Generated from item 'CurrentAngleLeft' *)
	fCurrentAngleLeft : LREAL;
	(* Generated from item 'CurrentAngleRight' *)
	fCurrentAngleRight : LREAL;
END_VAR
VAR
	{attribute 'no_copy'}
	PETML_DH10_M : POINTER TO ST_RT_MODEL_ETML_DH10_T;
END_VAR

{attribute 'TcTypeSystem'}

METHOD FB_exit : BOOL
VAR_INPUT
	bInCopyCode : BOOL;
END_VAR
END_METHOD

{attribute 'TcTypeSystem'}

METHOD FB_init : BOOL
VAR_INPUT
	bInitRetains : BOOL;
	bInCopyCode : BOOL;
END_VAR
END_METHOD

{attribute 'TcTypeSystem'}

{attribute 'monitoring' := 'call'}
	PROPERTY nHResult : HRESULT
GET
END_GET
END_PROPERTY

{attribute 'TcTypeSystem'}

{attribute 'monitoring' := 'call'}
	PROPERTY eInitExceptionHandling : E_FpExcptCtrlSetEx
GET
END_GET
SET
END_SET
END_PROPERTY

{attribute 'TcTypeSystem'}

{attribute 'monitoring' := 'call'}
	PROPERTY eUpdateExceptionHandling : E_FpExcptCtrlSetEx
GET
END_GET
SET
END_SET
END_PROPERTY

{attribute 'TcTypeSystem'}

{attribute 'monitoring' := 'call'}
	PROPERTY nExceptionCnt : ULINT
GET
END_GET
END_PROPERTY

{attribute 'TcTypeSystem'}

{attribute 'monitoring' := 'variable'}
	PROPERTY stActiveException : ST_ExceptionInfo
GET
END_GET
END_PROPERTY

{attribute 'TcTypeSystem'}

{attribute 'monitoring' := 'call'}
	PROPERTY bInitialized : BOOL
GET
END_GET
END_PROPERTY

{attribute 'TcTypeSystem'}

{attribute 'monitoring' := 'call'}
	PROPERTY bExecute : BOOL
GET
END_GET
SET
END_SET
END_PROPERTY

END_FUNCTION_BLOCK

// POUs/TcCOM Wrapper/FB_ETML_DH10_TcCOM_InitStruct

{attribute 'c++_compatible'}
{attribute 'external_name' := 'FB_ETML_DH10_TcCOM_InitStruct_GUID_AB1092F6_37B7_66ED_05C5_73810702BC38'}
{attribute 'TcIecLibraryType'}
{attribute 'call_after_init'}
{attribute 'reflection'}
FUNCTION_BLOCK FB_ETML_DH10_TcCOM_InitStruct
VAR
	{attribute 'hide'}
	{attribute 'no_copy'}
	{attribute 'GUID' := '18071995-0000-0000-0000-000000000018'}
	m_pData : PVOID;
	{attribute 'TcInitSymbol'}
	{attribute 'GUID' := '8007AE3B-86BB-40F2-B385-EF87FCC239A4'}
	eTraceLevelMaxFB : TcTraceLevel := TcTraceLevel.tlInfo;
	 {attribute 'hide'}
	_reserved1 : UDINT;
	{attribute 'hide'}
	{attribute 'instance-path'}
	{attribute 'noinit'}
	{attribute 'GUID' := '18071995-0000-0000-0000-0001000000FF'}
	sInstancePath : STRING(255);
	{attribute 'hide'}
	{attribute 'noinit'}
	{attribute 'GUID' := '18071995-0000-0000-0000-000000000019'}
	m_HResultLog : HRESULT;
	{attribute 'hide'}
	{attribute 'noinit'}
	{attribute 'GUID' := '18071995-0000-0000-0000-000000000019'}
	m_HResult : HRESULT;
	 {attribute 'hide'}
	_reserved2 : UINT_0_32;
	 {attribute 'hide'}
	_reserved3 : ARRAY [1..12] OF UINT_8_16;
	 {attribute 'hide'}
	_reserved4 : ARRAY [1..12] OF USINT;
END_VAR
VAR_INPUT
	stETML_DH10_U : ST_ETML_DH10_U_T;
END_VAR
VAR_OUTPUT
	stETML_DH10_Y : ST_ETML_DH10_Y_T;
END_VAR
VAR
	{attribute 'hide'}
	{attribute 'GUID' := '22276226-8561-82D3-24FD-532348FCDDE2'}
	_ipETML_DH10 : POINTER TO ITcETML_DH10;
	stInit : ST_FB_ETML_DH10_TcCOM_InitStruct;
END_VAR

{attribute 'TcTypeSystem'}

METHOD FB_init : BOOL
VAR_INPUT
	bInitRetains : BOOL;
	bInCopyCode : BOOL;
	{attribute 'GUID' := '0A68B9CB-5B03-1245-EDC2-65569CCA7EED'}
	stInit : REFERENCE TO ST_FB_ETML_DH10_TcCOM_InitStruct;
END_VAR
END_METHOD

{attribute 'TcTypeSystem'}

{attribute 'call_after_init'}
METHOD FB_afterinit : BOOL
END_METHOD

{attribute 'TcTypeSystem'}

METHOD Reinit : BOOL
VAR_INPUT
	{attribute 'GUID' := '0A68B9CB-5B03-1245-EDC2-65569CCA7EED'}
	stReInit : ST_FB_ETML_DH10_TcCOM_InitStruct;
END_VAR
END_METHOD

{attribute 'TcTypeSystem'}

METHOD FB_exit : BOOL
VAR_INPUT
	bInCopyCode : BOOL;
END_VAR
END_METHOD

{attribute 'TcTypeSystem'}

	PROPERTY eObjectState : TCOM_STATE
GET
END_GET
SET
END_SET
END_PROPERTY

{attribute 'TcTypeSystem'}

{attribute 'monitoring' := 'call'}
	PROPERTY nHResult : HRESULT
GET
END_GET
END_PROPERTY

{attribute 'TcTypeSystem'}

	PROPERTY ipTcComObject : ITComObject
GET
END_GET
END_PROPERTY

{attribute 'TcTypeSystem'}

	PROPERTY ipADI : ITcADI
GET
END_GET
END_PROPERTY

{attribute 'TcTypeSystem'}

	PROPERTY nTaskOid : OTCID
GET
END_GET
SET
END_SET
END_PROPERTY

{attribute 'TcTypeSystem'}

	PROPERTY nTaskPriority : UDINT
GET
END_GET
END_PROPERTY

{attribute 'TcTypeSystem'}

	PROPERTY nTaskCycleTimeNs : UDINT
GET
END_GET
END_PROPERTY

{attribute 'TcTypeSystem'}

	PROPERTY nTaskPort : UINT
GET
END_GET
END_PROPERTY

{attribute 'TcTypeSystem'}

	PROPERTY nTaskSortOrder : UDINT
GET
END_GET
SET
END_SET
END_PROPERTY

{attribute 'TcTypeSystem'}

	PROPERTY eTraceLevelMax : TcTraceLevel
GET
END_GET
SET
END_SET
END_PROPERTY

{attribute 'TcTypeSystem'}

	PROPERTY eModuleCaller : E_ModuleCaller
GET
END_GET
SET
END_SET
END_PROPERTY

{attribute 'TcTypeSystem'}

	PROPERTY eCallerVerification : E_CallerVerification
GET
END_GET
SET
END_SET
END_PROPERTY

{attribute 'TcTypeSystem'}

	PROPERTY eStepSizeAdaptation : E_StepSizeAdaptation
GET
END_GET
SET
END_SET
END_PROPERTY

{attribute 'TcTypeSystem'}

	PROPERTY eExecutionSequence : E_ExecutionSequence1
GET
END_GET
SET
END_SET
END_PROPERTY

{attribute 'TcTypeSystem'}

	PROPERTY bExecute : BOOL
GET
END_GET
SET
END_SET
END_PROPERTY

{attribute 'TcTypeSystem'}

	PROPERTY eAccessLockState : TCOM_STATE
GET
END_GET
SET
END_SET
END_PROPERTY

{attribute 'TcTypeSystem'}

	PROPERTY eInitExceptionHandling : E_FpExcptCtrlSet
GET
END_GET
SET
END_SET
END_PROPERTY

{attribute 'TcTypeSystem'}

	PROPERTY eUpdateExceptionHandling : E_FpExcptCtrlSetEx
GET
END_GET
SET
END_SET
END_PROPERTY

{attribute 'TcTypeSystem'}

	PROPERTY stModuleBuildInfo : ST_ModuleBuildInfo
GET
END_GET
END_PROPERTY

{attribute 'TcTypeSystem'}

	PROPERTY bInitialized : BOOL
GET
END_GET
END_PROPERTY

{attribute 'TcTypeSystem'}

	PROPERTY nSkippedExecutionCount : UDINT
GET
END_GET
END_PROPERTY

{attribute 'TcTypeSystem'}

	PROPERTY stLibraryInfo : ST_LibraryInfo
GET
END_GET
END_PROPERTY

{attribute 'TcTypeSystem'}

	PROPERTY stModuleInfo : ST_ModuleInfo
GET
END_GET
END_PROPERTY

{attribute 'TcTypeSystem'}

	PROPERTY stModuleGeneratorInfo : ST_TcMatSim_ModuleGeneratorInfo
GET
END_GET
SET
END_SET
END_PROPERTY

{attribute 'TcTypeSystem'}

	PROPERTY stSimulinkModelInfo : ST_TcMatSim_SimulinkModelInfo
GET
END_GET
SET
END_SET
END_PROPERTY

{attribute 'TcTypeSystem'}

	PROPERTY eETML_DH10_P_Sharing : E_ParameterSharingType
GET
END_GET
SET
END_SET
END_PROPERTY

{attribute 'TcTypeSystem'}

	PROPERTY nETML_DH10_P_Definer : OTCID
GET
END_GET
END_PROPERTY

{attribute 'TcTypeSystem'}

	PROPERTY stETML_DH10_P : ST_P_ETML_DH10_T
GET
END_GET
SET
END_SET
END_PROPERTY

{attribute 'TcTypeSystem'}

	PROPERTY nCycleCount : ULINT
GET
END_GET
END_PROPERTY

{attribute 'TcTypeSystem'}

	PROPERTY nExceptionCount : ULINT
GET
END_GET
END_PROPERTY

{attribute 'TcTypeSystem'}

	PROPERTY stExceptionInfo : ST_ExceptionInfo
GET
END_GET
END_PROPERTY

END_FUNCTION_BLOCK
